{attribute 'to_string'}
TYPE EN_BatchEvents :
(
	ALL				:= 0,
	RECIPE		    := 1,
	BATCH			:= 2,
	SETTINGS		:= 3,
	CALIBRATION		:= 4,
	ACTIONS			:= 5
);
END_TYPE

(* stored: Version 1.1.0.1, ProductVersion 3.1.4024.12
   DUT EN_BatchEvents: Id {e5c444a5-4ba3-42b6-9813-e5525bfa9fc4} *)
